FUNCTION ID_equal_to_ID : BOOL
VAR_INPUT
	ID1 :  REFERENCE TO Tag_ID;
	ID2 :  REFERENCE TO Tag_ID;
END_VAR

VAR CONSTANT 
	TagSize : UINT := 8;
END_VAR

VAR
	i : UINT;
	TagEqual : BOOL := TRUE;
END_VAR

FOR i:=0 TO TagSize-1 BY 1 DO
	TagEqual := TagEqual AND ID1[i] = ID2[i];
	// TODO Stop for loop waneer niet gelijk
END_FOR

ID_equal_to_ID := TagEqual;

END_FUNCTION

(* stored: Version 1.1.0.1, ProductVersion 3.1.4024.10
   POU ID_equal_to_ID: Id {eb2f5e9c-4573-433a-8055-6463937ca6ab}, SpecialFunc None *)
